// TIA Portal V16 export
// export: Created 2023-08-28T09:37:49.0816623Z, ExportSetting WithDefaults, DisplayName Totally Integrated Automation Portal, DisplayVersion V16 Update 6, DisplayName TIA Portal Version Control Interface, DisplayVersion V16 Update 2, DisplayName TIA Portal Openness, DisplayVersion V16 Update 6, DisplayName STEP 7 Professional, DisplayVersion V16 Update 6, DisplayName STEP 7 Safety, DisplayVersion V16, DisplayName WinCC Advanced, DisplayVersion V16 Update 6
DATA_BLOCK "dbcalculation_of_the_increment"   // DB18
AUTHOR : RTecmer
FAMILY : PID
VERSION : 0.1
// stored: AutoNumber true, DBAccessibleFromOPCUA true, InstanceOfName 07_E_Pressure build-up control, InstanceOfType FB
"07_E_Pressure build-up control"
   // VAR_INPUT
   //    "50Hz" : Bool;
   //    "Set_O2-PID" : Real;
   //    Current_bar_1 : Real;
   // END_VAR
   // VAR_OUTPUT
   //    Increase_in_value : Bool;
   // END_VAR
   // VAR_IN_OUT
   //    Edge1_Hz : Bool;
   //    Edge2_Hz : Bool;
   //    Data_sek_1 : Int;
   //    Data_sek_2 : Int;
   //    Pause_1 : Bool;
   //    Pause_2 : Bool;
   // END_VAR
BEGIN
END_DATA_BLOCK
